{attribute 'GeneratedUsingTerminal: EL5102-0000-0016'}
{attribute addProperty BoxType "EL5102-0000-0016"}
{attribute addProperty Id "StatusAT %I*Status_AA25F79C20Counter_valueAT %I*UDINT4Latch_valueAT %I*UDINT4Latch_value_2AT %I*UDINT4"}
{attribute addProperty CRC "279346770"}
{attribute addProperty Size "32"}
TYPE ENC_Status_Channel_10A67E52 EXTENDS InputBase_8311D824 :
STRUCT
	{attribute addProperty Name "Status"}
	Status AT %I* : Status_AA25F79C;
	{attribute addProperty Name "Counter_value"}
	Counter_value AT %I* : UDINT;
	{attribute addProperty Name "Latch_value"}
	Latch_value AT %I* : UDINT;
	{attribute addProperty Name "Latch_value_2"}
	Latch_value_2 AT %I* : UDINT;
END_STRUCT
END_TYPE

(* stored: Version 1.2.0.0, ProductVersion 3.1.4024.9
   DUT ENC_Status_Channel_10A67E52: Id {c52b1e80-a8fd-48fb-a2f3-f73843293ea4} *)
